// Mitsubishi GX Works2 project: Primeira etapa aula 04102023   PLC: Q03UDV

// task Task_01 (event TRUE, interval 0, priority 31): POU_01
// task Tarefa1 (event TRUE, interval 0, priority 31): 
// task ST_example2 (event TRUE, interval 0, priority 31): ST_example2

PROGRAM POU_01
END_PROGRAM

PROGRAM ST_example2
VAR
  iElemvar0 : ;  (* Elemento com variação *)
END_VAR
VAR CONSTANT
  iElem0 :  := 15;
  iElem1 :  := 4;
END_VAR
VAR
  iElemvar1 : ;  (* 15 *)
  aiTesteCriacaoArray : ARRAY [0..9] OF BOOL;
  fbBlinkerTesteST : LD_Examples_Esteira;
  fbTimerPulse : TP;
END_VAR
iDR[0]:=
(*Indicações conforme F1*)
ENO: MOD
aiTesteCriacaoArray
fbTimerPulse(IN:= ?BOOL? ,PT:= ?TIME? ,Q:= ?BOOL? ,ET:= ?TIME? );
END_PROGRAM

FUNCTION_BLOCK fbSum
VAR
  i_Elesum1 : INT;
  i_Elesum2 : INT;
END_VAR
(* structured ladder/FBD written out as ST: instructions are called as NAME(EN, inputs, outputs); _pN, _eN, _tN stand for wires *)
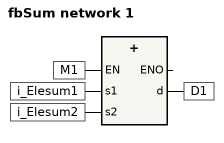
(* network 1 *)
+(M1, i_Elesum1, i_Elesum2, D1);
END_FUNCTION_BLOCK

FUNCTION_BLOCK fbSubtraction
VAR
  i_ElemSub1 : INT;
  i_ElemSub2 : INT;
END_VAR
(* structured ladder/FBD written out as ST: instructions are called as NAME(EN, inputs, outputs); _pN, _eN, _tN stand for wires *)
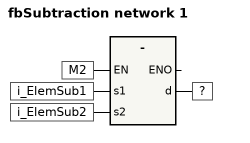
(* network 1 *)
-(M2, i_ElemSub1, i_ElemSub2, ?);
END_FUNCTION_BLOCK
